// TIA Portal V19 export
TYPE "LEXCHANGETRAY_typeRoller_deliver_interface_B2"
// stored: Access Published
   STRUCT
      init : Bool;
      logistics : "LEXCHANGETRAY_typeRoller_toLogisticsDeliver_B2";
      workStationRoller { S7_SetPoint := 'True'} : "LEXCHANGETRAY_typeRoller_toWorkstationDeliver_B2";
   END_STRUCT;
END_TYPE
